(* PLC project A2ServodriveLibrary, Delta Electronics, Inc. DIADesigner-AX DIADesigner-AX 1.3, author Piotr Gliszczyński *)
(* stored: creationDateTime 2022-10-25T14:05:01.3674589, version 3.5.15.30, modificationDateTime 2022-10-25T14:01:11.1788815, organization Induprogress sp. z o.o *)
(* Library for using A2 via CiA402. For now enum for error codes processing is available. *)

{attribute 'qualified_only'}
{attribute 'strict'}
TYPE DriveA2Error : (NO_ERROR := 0, OVER_CURRENT_AL001 := 16#1, OVER_VOLTAGE_AL002 := 16#2, UNDER_VOLTAGE_AL003 := 16#3, MOTOR_COMBINATION_ERROR_AL004 := 16#4, REGENERATION_ERROR_AL005 := 16#5, OVERLOAD_AL006 := 16#6, OVERSPEED_AL007 := 16#7, ABNORMAL_PULSE_COMMAND_AL008 := 16#8, EXCESSIVE_DEVIATION_OF_POSITION_COMMAND_AL009 := 16#9, ENCODER_ERROR_AL011 := 16#11, ADJUSTMENT_ERROR_AL012 := 16#12, EMERGENCY_STOP_AL013 := 16#13, REVERSE_LIMIT_ERROR_AL014 := 16#14, FORWARD_LIMIT_ERROR_AL015 := 16#15, IGBT_OVERHEAT_AL016 := 16#16, ABNORMAL_ERROR_AL017 := 16#17, ABNORMAL_SIGNAL_OUTPUT_AL018 := 16#18, SERIAL_COMMUNICATION_ERROR_AL019 := 16#19, SERIAL_COMMUNICATION_TIME_OUT_AL020 := 16#20, MAIN_CIRCUIT_POWER_LACK_PHASE_AL022 := 16#22, EARLY_WARNING_FOR_OVERLOAD_AL023 := 16#23, ENCODER_INITIAL_MAGNETIC_FIELD_ERROR_AL024 := 16#24, THE_INTERNAL_OF_THE_ENCODER_IS_IN_ERROR_AL025 := 16#25, UNRELIABLE_INTERNAL_DATA_OF_THE_ENCODER_AL026 := 16#26, THE_INTERNAL_OF_THE_IS_IN_ERROR_AL027 := 16#27, ENCODER_VOLTAGE_ERROR_AL028 := 16#28, GRAY_CODE_ERROR_AL029 := 16#29, MOTOR_CRASH_ERROR_AL030 := 16#30, INCORRECT_WIRING_OF_THE_MOTOR_POWER_LINE_UVW_GND_AL031 := 16#31, INTERNAL_COMMUNICATION_OF_THE_ENCODER_IS_IN_ERROR_AL034 := 16#34, ENCODER_TEMPERATURE_EXCEEDS_THE_PROTECTIVE_RANGE_AL035 := 16#35, EXCESSIVE_DEVIATION_OF_FULL_CLOSED_LOOP_AL040 := 16#40, COMMUNICATION_OF_LINEAR_SCALE_IS_BREAKDOWN_AL041 := 16#41, ANALOG_INPUT_VOLTAGE_ERROR_AL042 := 16#42, WARNING_OF_SERVODRIVE_FUNCTION_OVERLOAD_AL043 := 16#43, WRONG_SETTING_OF_E_GEAR_RATIO_AL045 := 16#45, THE_ABSOLUTE_POSITION_IS_LOST_AL060 := 16#60, ENCODER_UNDER_VOLTAGE_AL061 := 16#61, THE_MULTITURN_OF_ABSOLUTE_ENCODER_OVERFLOWS_AL062 := 16#62, ENCODER_TEMPERATURE_WARNING_AL067 := 16#67, ABSOLUTE_DATA_TRANSMITTED_VIA_IO_IS_IN_ERROR_AL068 := 16#68, WRONG_MOTOR_TYPE_AL069 := 16#69, THE_ABSOLUTE_COORDINATE_HAS_NOT_BEEN_INITIALIZED_AL06A := 16#6A, ENCODER_DOES_NOT_COMPLETE_THE_COMMAND_AL070 := 16#70, ENCODER_OVERSPEED_AL072 := 16#72, ENCODER_MEMORY_ERROR_AL073 := 16#73, ABSOLUTE_ENCODER_SINGLE_TURN_POSITION_ERROR_AL074 := 16#74, ABSOLUTE_ENCODER_POSITION_ERROR_AL075 := 16#75, ENCODER_COMPUTING_ERROR_AL077 := 16#77, ENCODER_PARAMETER_ERROR_AL079 := 16#79, LOSS_OF_ENCODER_Z_PULSE_AL07A := 16#7A, ENCODER_MEMORY_BUSY_AL07B := 16#7B, COMMAND_TO_CLEAR_THE_ABSOLUTE_POSITION_ISSUED_WHEN_MOTOR_SPEED_OVER_200_RPM_AL07C := 16#7C, SERVODRIVE_POWER_IS_CYCLED_BEFORE_AL07C_IS_CLEARED_AL07D := 16#7D, ENCODER_CLEARING_PROCEDURE_ERROR_AL07E := 16#7E, SERVO_DRIVE_OUTPUTS_EXCESSIVE_CURRENT_AL083 := 16#83, REGENERATION_SETTING_ERROR_AL085 := 16#85, INPUT_VOLTAGE_IS_TOO_HIGH_AL086 := 16#86, THE_SERVO_DRIVE_DOES_NOT_CONNECT_TO_EXTERNAL_REGENERATIVE_RESISTOR_AL095 := 16#95, DSP_FIRMWARE_UPGRADE_AL099 := 16#99, CANOPEN_SDO_RECIEVES_BUFFER_OVERFLOW_AL111 := 16#111, CANOPEN_PDO_RECIEVES_BUFFER_OVERFLOW_AL112 := 16#112, INDEX_ERROR_OCCURS_WHEN_ACCESING_CANOPEN_PDO_AL121 := 16#121, SUBINDEX_ERROR_OCCURS_WHEN_ACCESING_CANOPEN_PDO_AL122 := 16#122, DATA_SIZE_ERROR_OCCURS_WHEN_ACCESING_CANOPEN_PDO_AL123 := 16#123, DATA_RANGE_ERROR_OCCURS_WHEN_ACCESING_CANOPEN_PDO_AL124 := 16#124, CANOPEN_PDO_IS_READONLY_AND_WRITE_PROTECTED_AL125 := 16#125, CANOPEN_PDO_IS_NOT_ALLOWED_IN_PDO_AL126 := 16#126, CANOPEN_PDO_IS_WRITE_PROTECTED_WHEN_SERVO_ON_AL127 := 16#127, ERROR_OCCURS_WHEN_READING_CANOPEN_PDO_VIA_EEPROM_AL128 := 16#128, ERROR_OCCURS_WHEN_WRITING_CANOPEN_PDO_VIA_EEPROM_AL129 := 16#129, THE_ACCESSING_ADDRESS_OF_EEPROM_IS_OUT_OF_RANGE_WHEN_USING_CANOPEN_PDO_AL130 := 16#130, CRC_OF_EEPROM_CALCULATION_ERROR_OCCURS_WHEN_USING_CANOPEN_PDO_AL131 := 16#131, ENTER_THE_INCORRECT_PASSWORD_WHEN_USING_CANOPEN_PDO_AL132 := 16#132, HEARTBEAT_OR_NODEGUARDING_ERROR_AL170 := 16#170, CANOPEN_PDO_TIMEOUT_AL180 := 16#180, COMMUNICATION_DISCONNECTED_AL185 := 16#185, CAN_BUS_OFF_AL186 := 16#186, ERROR_OCCURS_WHEN_LOADING_CANOPEN_DATA_AL201 := 16#201, PARAMETER_GROUP_OF_PR8_IS_OUT_OF_RANGE_AL207 := 16#207, PARAMETER_NUMBER_OF_PR8_IS_OUT_OF_RANGE_AL209 := 16#209, PARAMETER_SETTING_OF_PR8_IS_WRONG_AL213 := 16#213, WRITE_PARAMETERS_READ_ONLY_AL215 := 16#215, WRITE_PARAMETERS_PARAMETERS_LOCKED_AL217 := 16#217, SETTING_OF_MONITOR_ITEM_OF_PR8_IS_OUT_OF_RANGE_AL231 := 16#231, PR_COMMAND_OVERFLOWS_AL235 := 16#235, INDEXING_COORDINATE_IS_UNDEFINED_AL237 := 16#237, PR_POSITIONING_TIMEOUT_AL245 := 16#245, THE_NUMBER_OF_PR_COMMAND_EXCEEDS_THE_LIMIT_AL249 := 16#249, FORWARD_SOFTWARE_LIMIT_AL283 := 16#283, REVERSE_SOFTWARE_LIMIT_AL285 := 16#285, FEEDBACK_POSITION_COUNTER_OVERFLOWS_AL289 := 16#289, SERVO_OFF_ERROR_AL291 := 16#291, CANOPEN_FAILS_TO_SYNCHRONIZE_AL301 := 16#301, THE_SYNCHRONIZED_SIGNAL_OF_CANOPEN_IS_SENT_TO_FAST_AL302 := 16#302, THE_SYNCHRONIZED_SIGNAL_OF_CANOPEN_IS_SENT_TOO_SLOW_AL303 := 16#303, CANOPEN_IP_COMMAND_IS_FAILED_AL304 := 16#304, SYNC_PERIOD_IS_IN_ERROR_AL305 := 16#305, EMERGENCY_STOP_DURING_DECELERATION_AL35F := 16#35F, POSITION_DEVIATION_ALARM_FOR_DO_MC_OK_AL380 := 16#380, EMERGENCY_STOP_AL3CF := 16#3CF, CANOPEN_SYNC_FAILED_SERVO_OFF_AL3E1 := 16#3E1, CANOPEN_SYNC_SIGNAL_ERROR_SERVO_OFF_AL3E2 := 16#3E2, CANOPEN_SYNC_TIME_OUT_AL3E3 := 16#3E3, CANOPEN_IP_COMMAND_FAILED_AL3E4 := 16#3E4, SYNC_PERIOD_ERROR_AL3E5 := 16#3E5, ABSOLUTE_INDEX_COORDINATE_UNDEFINED_AL3F1 := 16#3F1, INDEX_COORDINATES_ERROR_AL400 := 16#400, NMT_RESET_COMMAND_IS_RECIEVED_WHEN_SERVO_ON_AL401 := 16#401, VALUE_OF_PR_SPECIAL_FILTER_SETTING_IS_TOO_BIG_AL404 := 16#404, SAFE_TORQUE_ENABLED_AL500 := 16#500, STO_A_LOSS_AL501 := 16#501, STO_B_LOSS_AL502 := 16#502, STO_SELF_DIAGNOSTIC_ERROR_AL503 := 16#503, SYSTEM_FAILURE_AL555 := 16#555);
END_TYPE
